// TIA Portal V20 export
DATA_BLOCK "ManualOperationControl_U1Em5"   // DB22
// stored: MemoryReserve 100
   VAR
      manualOperationEm { ExternalAccessible := 'False'; ExternalVisible := 'False'; ExternalWritable := 'False'} : "LAF_typeManEm";
      manualOperationEmArea { ExternalAccessible := 'False'; ExternalVisible := 'False'; ExternalWritable := 'False'} : Array[1..2] of "LAF_typeManOperationArea";
      manualOperationCms { ExternalAccessible := 'False'; ExternalVisible := 'False'; ExternalWritable := 'False'} : Array[1..90] of "LAF_typeManOperation";
      axis { S7_SetPoint := 'True'} : Array[0..6] of "LBC_typeAxis64PosInterface";
      softCam { S7_SetPoint := 'True'} : Array[0..20] of "LER_typeSoftCamRelation";
      twoWayActuator { S7_SetPoint := 'True'} : Array[0..2] of "LBC_typeTwoWayActuatorInterface";
   END_VAR
BEGIN
   manualOperationEm.equipmentModuleNum := 1060;
   manualOperationEmArea[1].displayedLines := '1';
END_DATA_BLOCK
